(*Used as soft IO mapping to creat a psuedo gague to communicate over two taks on the same PLC.*) 
(*for FAST shutter control*)
FUNCTION_BLOCK FB_GFS_Interface
VAR_INPUT
	IG : ST_VG; // The Cold Cathode Data Structure
END_VAR
VAR_OUTPUT
END_VAR
VAR
	(*inputs*)
	{attribute 'pytmc' := '
	pv: TRIG; 
	field: ZNAM TRIG_OFF; 
	field: ONAM TRIG_ON;
	io: io ;
	'}
	i_xTrigger AT %I* : BOOL;
	{attribute 'pytmc' := '
	pv: OPEN; 
	field: ZNAM NOT OPEN; 
	field: ONAM OPEN;
	io: io ;
	'}
	i_xVFS_Open AT %I* : BOOL;
	{attribute 'pytmc' := '
	pv: CLS; 
	field: ZNAM NOT CLOSED; 
	field: ONAM CLOSE;
	io: io ;
	'}
	i_xVFS_Closed AT %I* : BOOL;
	{attribute 'pytmc' := '
	pv: FAULT_OK; 
	field: ZNAM FAULT ; 
	field: ONAM FAULT OK;
	io: io ;
	'}
	xVAC_FAULT_OK AT%Q*: BOOL; (*Valve Vacuum OK, is set to False when there is Vacuum Fault*)

	(*outputs*)
	q_xPRESS_OK AT%Q*: BOOL;
END_VAR


(*soft IO Mapping*)

q_xPRESS_OK := IG.xPRESS_OK;

END_FUNCTION_BLOCK

(* stored: Version 1.1.0.1, ProductVersion 3.1.4022.16
   POU FB_GFS_Interface: Id {781a56cb-c763-46ed-9ac5-b2e690be9ff4}, SpecialFunc None *)
